                   REGION "SOLID RED"
                       IF #animation = #anSolidRed THEN
                           CASE #j OF
                               #"Part 01":
                                   #stackLight := #stackLight OR #"Part 01 Red On";
                                   #stackLight := #stackLight AND (NOT #"Part 01 Yellow On");
                                   #stackLight := #stackLight AND (NOT #"Part 01 Green On");
                               #"Part 02":
                                   #stackLight := #stackLight OR #"Part 02 Red On";
                                   #stackLight := #stackLight AND (NOT #"Part 02 Yellow On");
                                   #stackLight := #stackLight AND (NOT #"Part 02 Green On");
                               #"Part 03":
                                   #stackLight := #stackLight OR #"Part 03 Red On";
                                   #stackLight := #stackLight AND (NOT #"Part 03 Yellow On");
                                   #stackLight := #stackLight AND (NOT #"Part 03 Green On");
                               #"Part 04":
                                   #stackLight := #stackLight OR #"Part 04 Red On";
                                   #stackLight := #stackLight AND (NOT #"Part 04 Yellow On");
                                   #stackLight := #stackLight AND (NOT #"Part 04 Green On");
                               #"Part 05":
                                   #stackLight := #stackLight OR #"Part 05 Red On";
                                   #stackLight := #stackLight AND (NOT #"Part 05 Yellow On");
                                   #stackLight := #stackLight AND (NOT #"Part 05 Green On");
                               #"Part 06":
                                   #stackLight := #stackLight OR #"Part 06 Red On";
                                   #stackLight := #stackLight AND (NOT #"Part 06 Yellow On");
                                   #stackLight := #stackLight AND (NOT #"Part 06 Green On");
                               ELSE
                                   ;
                           END_CASE;
                       END_IF;
                   END_REGION

                   REGION "FLASHING RED"
                       IF #animation = #anFlashRed THEN

                           REGION "RED ON"
                               IF "Clock_1Hz" THEN
                                   CASE #j OF
                                       #"Part 01":
                                           #stackLight := #stackLight OR #"Part 01 Red On";
                                           #stackLight := #stackLight AND (NOT #"Part 01 Yellow On");
                                           #stackLight := #stackLight AND (NOT #"Part 01 Green On");
                                       #"Part 02":
                                           #stackLight := #stackLight OR #"Part 02 Red On";
                                           #stackLight := #stackLight AND (NOT #"Part 02 Yellow On");
                                           #stackLight := #stackLight AND (NOT #"Part 02 Green On");
                                       #"Part 03":
                                           #stackLight := #stackLight OR #"Part 03 Red On";
                                           #stackLight := #stackLight AND (NOT #"Part 03 Yellow On");
                                           #stackLight := #stackLight AND (NOT #"Part 03 Green On");
                                       #"Part 04":
                                           #stackLight := #stackLight OR #"Part 04 Red On";
                                           #stackLight := #stackLight AND (NOT #"Part 04 Yellow On");
                                           #stackLight := #stackLight AND (NOT #"Part 04 Green On");
                                       #"Part 05":
                                           #stackLight := #stackLight OR #"Part 05 Red On";
                                           #stackLight := #stackLight AND (NOT #"Part 05 Yellow On");
                                           #stackLight := #stackLight AND (NOT #"Part 05 Green On");
                                       #"Part 06":
                                           #stackLight := #stackLight OR #"Part 06 Red On";
                                           #stackLight := #stackLight AND (NOT #"Part 06 Yellow On");
                                           #stackLight := #stackLight AND (NOT #"Part 06 Green On");
                                       ELSE
                                           ;
                                   END_CASE;
                               END_IF;
                           END_REGION

                           REGION "RED OFF"
                               IF NOT "Clock_1Hz" THEN
                                   CASE #j OF
                                       #"Part 01":
                                           #stackLight := #stackLight AND (NOT #"Part 01 Red On");
                                           #stackLight := #stackLight AND (NOT #"Part 01 Yellow On");
                                           #stackLight := #stackLight AND (NOT #"Part 01 Green On");
                                       #"Part 02":
                                           #stackLight := #stackLight AND (NOT #"Part 02 Red On");
                                           #stackLight := #stackLight AND (NOT #"Part 02 Yellow On");
                                           #stackLight := #stackLight AND (NOT #"Part 02 Green On");
                                       #"Part 03":
                                           #stackLight := #stackLight AND (NOT #"Part 03 Red On");
                                           #stackLight := #stackLight AND (NOT #"Part 03 Yellow On");
                                           #stackLight := #stackLight AND (NOT #"Part 03 Green On");
                                       #"Part 04":
                                           #stackLight := #stackLight AND (NOT #"Part 04 Red On");
                                           #stackLight := #stackLight AND (NOT #"Part 04 Yellow On");
                                           #stackLight := #stackLight AND (NOT #"Part 04 Green On");
                                       #"Part 05":
                                           #stackLight := #stackLight AND (NOT #"Part 05 Red On");
                                           #stackLight := #stackLight AND (NOT #"Part 05 Yellow On");
                                           #stackLight := #stackLight AND (NOT #"Part 05 Green On");
                                       #"Part 06":
                                           #stackLight := #stackLight AND (NOT #"Part 06 Red On");
                                           #stackLight := #stackLight AND (NOT #"Part 06 Yellow On");
                                           #stackLight := #stackLight AND (NOT #"Part 06 Green On");
                                       ELSE
                                           ;
                                   END_CASE;
                               END_IF;
                           END_REGION

                       END_IF;
                   END_REGION

                   REGION "COPY OUT TO GLOBAL"
                       #stations.current[#i].stackLightOut := #stackLight;
                   END_REGION

               END_FOR;
           END_REGION

       END_FOR;
   END_REGION
END_FUNCTION_BLOCK

FUNCTION_BLOCK "KP8 Button Activation"   // FB12, SCL
{ S7_Optimized_Access := 'TRUE' }
VERSION : 0.1
   VAR_INPUT
      constants : "Constants";
   END_VAR
   VAR_IN_OUT
      stations : "Stations";
   END_VAR
   VAR_TEMP
      btnCount : Int;
      currentPNs : Array[0..7] of WString[40];
      i : Int;
      init : Bool;
      j : Int;
      stnCount : Int;
      temp : Int;
   END_VAR
BEGIN
   REGION "GET STATION COUNT"
       #stnCount := #constants.stationCount - 1;
       #btnCount := #constants.buttonCount - 1;
   END_REGION

   REGION "LOOP THROUGH STATIONS"
       FOR #i := 0 TO #stnCount DO

           #currentPNs := #stations.current[#i].partNumbers;

           REGION "LOOP THROUGH BUTTONS"
               FOR #j := 0 TO #btnCount DO

                       REGION "ACTIVATE BUTTON"
                           IF LEN(#currentPNs[#j]) <> 0 THEN
                               #stations.current[#i].kp8Config.activate[#j] := TRUE;
                               #stations.current[#i].kp8Config.colorOff[#j] := 'green';
                               #stations.current[#i].kp8Config.colorOn1[#j] := 'yellow';
                               #stations.current[#i].kp8Config.colorOn2[#j] := '';
                               #stations.current[#i].kp8Config.flash[#j] := FALSE;
                               #stations.current[#i].kp8Config.group[#j] := 0;
                               #stations.current[#i].kp8Config.mode[#j] := TRUE;
                           END_IF;
                       END_REGION

                       REGION "DEACTIVATE BUTTON"
                           IF LEN(#currentPNs[#j]) = 0 THEN
                               #stations.current[#i].kp8Config.activate[#j] := FALSE;
                               #stations.current[#i].kp8Config.colorOff[#j] := '';
                               #stations.current[#i].kp8Config.colorOn1[#j] := '';
                               #stations.current[#i].kp8Config.colorOn2[#j] := '';
                               #stations.current[#i].kp8Config.flash[#j] := FALSE;
                               #stations.current[#i].kp8Config.group[#j] := 0;
                               #stations.current[#i].kp8Config.mode[#j] := FALSE;
                           END_IF;
                       END_REGION

               END_FOR;
           END_REGION

           REGION "SOFT INIT"
               IF #stations.current[#i].kp8Config <> #stations.old[#i].kp8Config THEN
                   #stations.current[#i].init.soft := TRUE;
               END_IF;
           END_REGION

       END_FOR;
   END_REGION
END_FUNCTION_BLOCK

FUNCTION_BLOCK "Remove Part Request"   // FB13, SCL
{ S7_Optimized_Access := 'TRUE' }
VERSION : 0.1
   VAR_INPUT
      constants : "Constants";
   END_VAR
   VAR_IN_OUT
      pRow : Int;
      requests : "Part Request Data";
      stations : "Stations";
   END_VAR
   VAR_TEMP
      address : UInt;
      blankRow : "Table Row";
      hasPart : Bool;
      i : Int;
      j : Int;
      k : Int;
      logAddress : UInt;
      maxRows : Int;
      noPart : Bool;
      oldPartReq : Bool;
      partNumber : WString;
      partReq : Bool;
      pRemoveRow : Int;
      btnCount : Int;
      stnCount : Int;
      removeAddress : Bool;
   END_VAR
BEGIN
   REGION "COPY TO LOCAL"
       #maxRows := #constants.partReqRows - 1;
       #stnCount := #constants.stationCount - 1;
       #btnCount := #constants.buttonCount - 1;
   END_REGION


   REGION "LOOP THROUGH STATIONS"
       FOR #i := 0 TO #stnCount DO

           REGION "LOOP THROUGH BUTTONS"
               FOR #j := 1 TO #btnCount DO

                   REGION "PRE-CONDITION"
                       // copy bits for falling edge detection
                       #partReq := #stations.current[#i].btnStates[#j];
                       #oldPartReq := #stations.old[#i].btnStates[#j];
                   END_REGION

                   REGION "DETERMINE STATE"
                       // falling edge detection
                       IF NOT #partReq AND #oldPartReq THEN
                           // copy to local
                           #partNumber := #stations.current[#i].partNumbers[#j];
                           // no part
                           IF #partNumber = wstring#'' THEN
                               #hasPart := FALSE;
                               #noPart := TRUE;
                           END_IF;
                           // has part
                           IF #partNumber <> wstring#'' THEN
                               #hasPart := TRUE;
                               #noPart := FALSE;
                           END_IF;
                       END_IF;
                   END_REGION

                   REGION "NO PART"
                       IF #noPart THEN
                           // turn off the lights
                           #hasPart := FALSE;
                           #noPart := FALSE;
                       END_IF;

                   END_REGION

                   REGION "HAS PART"
                       IF #hasPart THEN
                           // turn off the lights
                           #hasPart := FALSE;
                           // calculate address
                           #address := (INT_TO_UINT(#i) + 1) * 10 + (INT_TO_UINT(#j) + 1);
                           // precondition remove address flag
                           #removeAddress := FALSE;
                           // check table for previous entry
                           FOR #k := 0 TO #maxRows DO
                               #logAddress := #requests.row[#k].address;
                               // remove matching address flag
                               IF #logAddress = #address THEN
                                   #removeAddress := TRUE;
                                   #pRemoveRow := #k;
                               END_IF;
                           END_FOR;
                       END_IF;
                   END_REGION

                   REGION "REMOVE ADDRESS"
                       IF #removeAddress THEN

                           // turn off the lights
                           #removeAddress := FALSE;

                           REGION "REMOVAL PROCESS"
                               #requests.row[#pRemoveRow] := #blankRow;
                           END_REGION

                           REGION "ADJUST TABLE BLANK ROW POINTER"
                               // decriment row pointer
                               #pRow := #pRow - 1;
                               IF #pRow < 0 THEN
                                   #pRow := 0;
                               END_IF;
                           END_REGION

                       END_IF;
                   END_REGION

               END_FOR;

           END_REGION

       END_FOR;
   END_REGION
END_FUNCTION_BLOCK

FUNCTION_BLOCK "HMI Settings Screen"   // FB14, LAD
{ S7_Optimized_Access := 'TRUE' }
VERSION : 0.1
   VAR_INPUT
      constants : "Constants";
   END_VAR
   VAR_IN_OUT
      settings : "Settings Screen";
      stations : "Stations";
   END_VAR
   VAR
      tmrTimeOut : TON_TIME;
      instStaSel : "Station Selection";
      instKP8BtnSel : "KP8 Button Selections";
      instStnDetails : "Station Details";
   END_VAR
   VAR CONSTANT
      ptTimeOut : Time := t#15m;
   END_VAR
BEGIN

REGION Network 1: ENTRY TIMEOUT
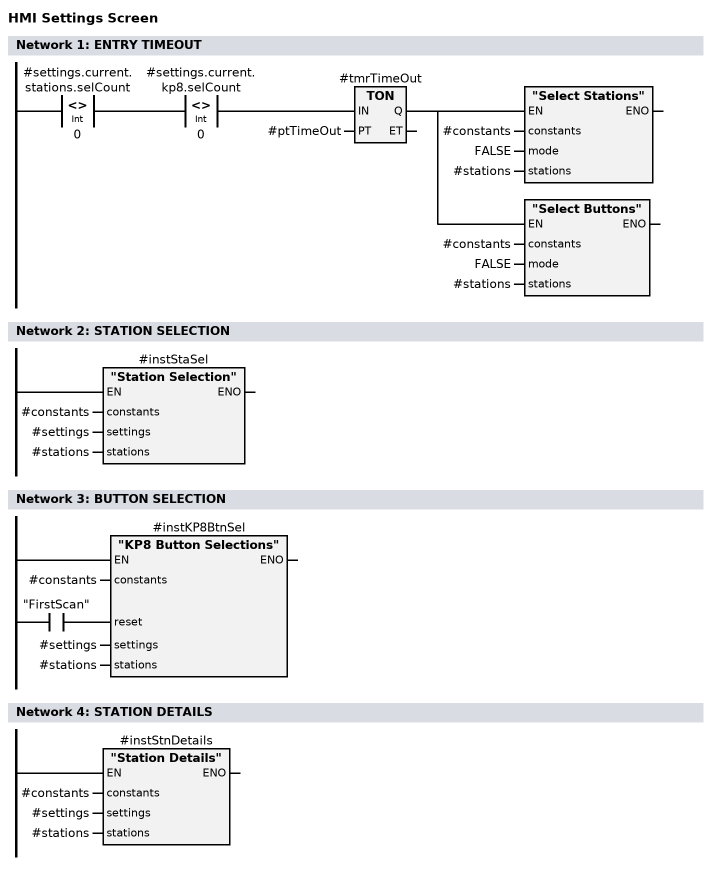
   #tmrTimeOut(IN := (#settings.current.stations.selCount <> 0) AND (#settings.current.kp8.selCount <> 0),   // TON
               PT := #ptTimeOut);
   IF #tmrTimeOut.Q THEN
       "Select Stations"(constants := #constants, mode := FALSE, stations := #stations);
       "Select Buttons"(constants := #constants, mode := FALSE, stations := #stations);
   END_IF;
END_REGION

REGION Network 2: STATION SELECTION
   RUNG wire#powerrail
      #instStaSel(constants := #constants, settings := #settings, stations := #stations)
   END_RUNG
   // the same network as SCL:
   #instStaSel(constants := #constants, settings := #settings, stations := #stations);   // "Station Selection"
END_REGION

REGION Network 3: BUTTON SELECTION
   RUNG wire#powerrail
      #instKP8BtnSel(reset := wire#w1, constants := #constants, settings := #settings, stations := #stations)
   END_RUNG
   RUNG wire#powerrail
      Contact( "FirstScan" )
   END_RUNG wire#w1
   // the same network as SCL:
   #instKP8BtnSel(constants := #constants, reset := "FirstScan", settings := #settings, stations := #stations);   // "KP8 Button Selections"
END_REGION

REGION Network 4: STATION DETAILS
   RUNG wire#powerrail
      #instStnDetails(constants := #constants, settings := #settings, stations := #stations)
   END_RUNG
   // the same network as SCL:
   #instStnDetails(constants := #constants, settings := #settings, stations := #stations);   // "Station Details"
END_REGION
END_FUNCTION_BLOCK

FUNCTION_BLOCK "Collapse Table"   // FB15, SCL
{ S7_Optimized_Access := 'TRUE' }
VERSION : 0.1
   VAR_INPUT
      constants : "Constants";
   END_VAR
   VAR_IN_OUT
      requests : "Part Request Data";
   END_VAR
   VAR
      tableBox : "Part Request Data";
   END_VAR
   VAR_TEMP
      blankRow : "Table Row";
      collapseReq : Bool;
      i : Int;
      maxRows : Int;
      pCollapse : Int;
   END_VAR
BEGIN
   REGION "COPY TO LOCAL"
       #maxRows := #constants.partReqRows - 1;
   END_REGION

   REGION "REMOVE EMPTY ROWS"
       FOR #i := 0 TO #maxRows DO

           REGION "ROW IS NOT EMPTY"
               IF #requests.row[#i].address <> 0 THEN

                   REGION "MOVE TO TEMP TABLE"
                       #tableBox.row[#pCollapse] := #requests.row[#i];
                   END_REGION

                   REGION "POINTERS AND FLAGS"
                       #pCollapse := #pCollapse + 1;
                       #collapseReq := TRUE;
                   END_REGION

               END_IF;
           END_REGION

       END_FOR;
   END_REGION

   REGION "COLLAPSE TABLE"
       IF #collapseReq THEN

           REGION "TURN OFF THE LIGHTS"
               #collapseReq := FALSE;
           END_REGION

           REGION "COPY TEMP TO PERMANENT"
               #requests := #tableBox;
           END_REGION

           REGION "CLEAR VALUES FROM TEMP TABLE"
               FOR #i := 0 TO #maxRows DO
                   #tableBox.row[#i] := #blankRow;
               END_FOR;
           END_REGION
       END_IF;

   END_REGION
END_FUNCTION_BLOCK

FUNCTION_BLOCK "HMI Populate Part Call"   // FB16, SCL
{ S7_Optimized_Access := 'TRUE' }
VERSION : 0.1
   VAR_INPUT
      constants : "Constants";
      requests : "Part Request Data";
   END_VAR
   VAR_IN_OUT
      partCall : "Part Call Screen";
   END_VAR
   VAR
      pDisplay : Int;
   END_VAR
   VAR_TEMP
      firstRow : Int;
      i : Int;
      lastRow : Int;
      maxRows : Int;
      pRow : Int;
      visibleRows : Int;
      thisRow : Int;
   END_VAR
BEGIN
   #visibleRows := #constants.hmiRowCount - 1;
   #maxRows := #constants.partReqRows - 1;
   #firstRow := 0;
   #lastRow := #firstRow + #visibleRows;

   FOR #i := 0 TO #visibleRows DO
       #partCall.current[#i] := #requests.row[#i];
   END_FOR;
END_FUNCTION_BLOCK

FUNCTION_BLOCK "Clear Part Requests"   // FB17, SCL
{ S7_Optimized_Access := 'TRUE' }
VERSION : 0.1
   VAR_INPUT
      constants : "Constants";
      clearRequest : Bool;
   END_VAR
   VAR_IN_OUT
      requests : "Part Request Data";
      partCall : "Part Call Screen";
   END_VAR
   VAR_TEMP
      blankRow : "Table Row";
      i : Int;
      maxRows : Int;
   END_VAR
BEGIN
   REGION "ON REQUEST"
       IF #clearRequest THEN

           REGION "CLEAR HMI TABLE"
               #maxRows := #constants.hmiRowCount - 1;
               FOR #i := 0 TO #maxRows DO
                   #partCall.current[#i] := #blankRow;
               END_FOR;
           END_REGION

           REGION "CLEAR PART REQUEST DATA BASE"
               #maxRows := #constants.partReqRows - 1;
               FOR #i := 0 TO #maxRows DO
                   #requests.row[#i] := #blankRow;
               END_FOR;
           END_REGION

       END_IF;
   END_REGION
END_FUNCTION_BLOCK

FUNCTION_BLOCK "Load Default Timer Presets"   // FB18, SCL
{ S7_Optimized_Access := 'TRUE' }
VERSION : 0.1
   VAR_INPUT
      constants : "Constants";
      req : Bool;
   END_VAR
   VAR_IN_OUT
      stations : "Stations";
   END_VAR
   VAR
      oldReq : Bool;
   END_VAR
   VAR_TEMP
      alotted : Real;
      btnCount : Int;
      critical : Real;
      i : Int;
      j : Int;
      stnCount : Int;
      partNumber : WString;
   END_VAR
BEGIN
   REGION "COPY TO LOCAL"
       #alotted := #constants.defaultAlotted;
       #btnCount := #constants.buttonCount - 1;
       #critical := #constants.defaultCritical;
       #stnCount := #constants.stationCount - 1;
   END_REGION

   REGION "ON REQUEST RISING EDGE"
       IF #req AND NOT #oldReq THEN

           REGION "LOOP THROUGH STATIONS" 
               FOR #i := 0 TO #stnCount DO

                   REGION "LOOP THROUGH BUTTONS"
                       FOR #j := 0 TO #btnCount DO

                           REGION "IF BUTTON HAS ASSOCIATED PN"
                               #partNumber := #stations.current[#i].partNumbers[#j];
                               IF LEN(#partNumber) <> 0 THEN

                                   REGION "ASSIGN PRESET VALUES"
                                       #stations.current[#i].presetTime.allotted[#j] := #alotted;
                                       #stations.current[#i].presetTime.critical[#j] := #critical;
                                   END_REGION

                               END_IF;
                           END_REGION

                       END_FOR;
                   END_REGION

               END_FOR;
           END_REGION

       END_IF;
   END_REGION

   REGION "CHANGE DETECTION"
       #oldReq := #req;
   END_REGION ;
END_FUNCTION_BLOCK

FUNCTION_BLOCK "LED Populate Sign"   // FB19, SCL
{ S7_Optimized_Access := 'TRUE' }
VERSION : 0.1
   VAR_INPUT
      constants : "Constants";
      requests : "Part Request Data";
   END_VAR
   VAR_IN_OUT
      ledData : "LED Sign Data";
   END_VAR
   VAR_TEMP
      i : Int;
      visibleRows : Int;
   END_VAR
BEGIN
   REGION "COPY TO LOCAL"
       #visibleRows := #constants.ledRowCount - 1;
   END_REGION

   REGION "POPULATE SIGN DATA"
       FOR #i := 0 TO #visibleRows DO
           #ledData.row[#i] := #requests.row[#i];
       END_FOR;
   END_REGION
END_FUNCTION_BLOCK

FUNCTION_BLOCK "Station Selection"   // FB20, SCL
{ S7_Optimized_Access := 'TRUE' }
VERSION : 0.1
   VAR_INPUT
      constants : "Constants";
   END_VAR
   VAR_IN_OUT
      settings : "Settings Screen";
      stations : "Stations";
   END_VAR
   VAR
      firstStn : Int;
      rt : "Runtime Data";
      selectionExe : Bool;
      old : Struct
         prevGrp : Bool;
         nextGrp : Bool;
         stnSlct : Array[0..11] of Bool;
      END_STRUCT;
   END_VAR
   VAR_TEMP
      animate : USInt;
      btnPress : Bool;
      count : Int;
      currentBtn : Bool;
      evalObjCount : Int;
      i : Int;
      oldBtn : Bool;
      pStn : Int;
      stnCount : Int;
      stnName : WString;
      stnSelected : Bool;
      selState : Bool;
      timerExpired : Bool;
      stnSelLblCount : Int;
   END_VAR
   VAR CONSTANT
      ptTimer : Real := 1.5;
   END_VAR
BEGIN
   REGION "UI INTERACTION ANIMATIONS"

       REGION "NEXT GROUP"
           #btnPress := #settings.current.stations.nextGroup.actuate;
           #animate := "Animate Bool"(colorTrue := #constants.colorLib.BgLGr,
                                      colorFalse := #constants.colorLib.BgGray,
                                      evalSignal := #btnPress);
           #settings.current.stations.nextGroup.animate := #animate;
       END_REGION

       REGION "PREVIOUS GROUP"
           #btnPress := #settings.current.stations.prevGroup.actuate;
           #animate := "Animate Bool"(colorTrue := #constants.colorLib.BgLGr,
                                      colorFalse := #constants.colorLib.BgGray,
                                      evalSignal := #btnPress);
           #settings.current.stations.prevGroup.animate := #animate;
       END_REGION

       REGION "SELECT ALL STATIONS"
           #btnPress := #settings.current.stations.selectAll.actuate;
           #animate := "Animate Bool"(colorTrue := #constants.colorLib.BgLGr,
                                      colorFalse := #constants.colorLib.BgGray,
                                      evalSignal := #settings.current.stations.selectAll.actuate);
           #settings.current.stations.selectAll.animate := #animate;
       END_REGION

   END_REGION

   REGION "POPULATE STATION LABELS"

       REGION "PROCESS NEXT GROUP PRESS"

           REGION "COPY TO LOCAL"
               #stnCount := #constants.stationCount - 1;
               #currentBtn := #settings.current.stations.nextGroup.actuate;
               #oldBtn := #old.nextGrp;
           END_REGION

           REGION "FALLING EDGE OF NEXT GROUP"
               IF NOT #currentBtn AND #oldBtn THEN

                   REGION "INCREMENT FIRST STATION"
                       #firstStn := #firstStn + 2;
                   END_REGION

                   REGION "UPPER LIMIT ROLL OVER"
                       IF #firstStn > #stnCount THEN
                           #firstStn := #firstStn - #stnCount - 1;
                       END_IF;
                   END_REGION

               END_IF;
           END_REGION

           REGION "NEXT GROUP CHANGE DETECTION"
               #old.nextGrp := #currentBtn;
           END_REGION

       END_REGION

       REGION "PROCESS PREVIOUS GROUP PRESS"

           REGION "COPY TO LOCAL"
               #currentBtn := #settings.current.stations.prevGroup.actuate;
               #oldBtn := #old.prevGrp;
               #stnCount := #constants.stationCount - 1;
           END_REGION

           REGION "FALLING EDGE OF PREVIOUS GROUP"
               IF NOT #currentBtn AND #oldBtn THEN

                   REGION "DECREMENT FIRST STATION"
                       #firstStn := #firstStn - 2;
                   END_REGION

                   REGION "LOWER LIMIT ROLL OVER"
                       IF #firstStn < 0 THEN
                           #firstStn := #firstStn + #stnCount + 1;
                       END_IF;
                   END_REGION

               END_IF;
           END_REGION

           REGION "PREVIOUS GROUP CHANGE DETECTION"
               #old.prevGrp := #currentBtn;
           END_REGION

       END_REGION

       REGION "WRITE LABEL"

           REGION "COPY TO LOCAL"
               #evalObjCount := #constants.hmiSelStnCount - 1;
               #stnCount := #constants.stationCount - 1;
           END_REGION

           REGION "FOR EACH STATION SELECTION BUTTON"
               FOR #i := 0 TO #evalObjCount DO

                   REGION "CALCULATE POINTER"
                       #pStn := #firstStn + #i;
                   END_REGION

                   REGION "UPPER LIMIT ROLL OVER"
                       IF #pStn > #stnCount THEN
                           #pStn := #firstStn + #i - #stnCount - 1;
                       END_IF;
                   END_REGION

                   REGION "BUILD NAME"
                       #stnName := CONCAT_WSTRING(IN1 := #stations.current[#pStn].line,
                                                  IN2 := wstring#' ',
                                                  IN3 := "Strip Sign"(USINT_TO_WSTRING(#stations.current[#pStn].dropZone)));
                   END_REGION

                   REGION "WRITE NAME"
                       #settings.current.stations.selectBtns[#i].label := #stnName;
                   END_REGION

               END_FOR;
           END_REGION

       END_REGION

   END_REGION

   REGION "SINGLE STATION SELECTION"

       REGION "COPY TO LOCAL"
           #stnSelLblCount := #constants.hmiSelStnCount - 1;
       END_REGION

       REGION "LOOP THROUGH DISPLAYED STATIONS"
           FOR #i := 0 TO #stnSelLblCount DO

               REGION "CALCULATE POINTER"
                   #pStn := #firstStn + #i;
               END_REGION

               REGION "UPPER LIMIT ROLL OVER"
                   #stnCount := #constants.stationCount - 1;
                   IF #pStn > #stnCount THEN
                       #pStn := #firstStn + #i - #stnCount - 1;
                   END_IF;
               END_REGION

               REGION "COPY TO LOCAL"
                   #currentBtn := #settings.current.stations.selectBtns[#i].actuate;
                   #oldBtn := #old.stnSlct[#i];
               END_REGION

               REGION "TOGGLE STATE ON FALLING EDGE"
                   IF NOT #currentBtn AND #oldBtn THEN
                       #selState := #stations.current[#pStn].settings.selected;
                       #selState := NOT #selState;
                       #stations.current[#pStn].settings.selected := #selState;
                   END_IF;
               END_REGION

               REGION "STATION SELECTION CHANGE DETECTION"
                   #old.stnSlct[#i] := #currentBtn;
               END_REGION

           END_FOR;
       END_REGION

   END_REGION

   REGION "MULTI SELECT TIMER"

       REGION "RUNTIME CALL"
           #rt.elapsed := RUNTIME(#rt.mem);
       END_REGION

       REGION "TIMER"

           REGION "COPY TO LOCAL"
               #btnPress := #settings.current.stations.selectAll.actuate;
           END_REGION

           REGION "ACCUMULATE RT VALUES"
               IF #btnPress THEN
                   #rt.asReal += LREAL_TO_REAL(#rt.elapsed);
               END_IF;
           END_REGION

           REGION "SET TIMER FLAG"
               IF #rt.asReal < #ptTimer THEN
                   #timerExpired := FALSE;
               END_IF;
               IF #rt.asReal >= #ptTimer THEN
                   #timerExpired := TRUE;
                   #rt.asReal := 0.0;
               END_IF;
           END_REGION

           REGION "RESET ACCUMULATED VALUE"
               IF NOT #btnPress THEN
                   #rt.asReal := 0.0;
                   #selectionExe := FALSE;
               END_IF;
           END_REGION

       END_REGION

   END_REGION

   REGION "EVALUATE MULTI SELECTION"
       IF #timerExpired AND NOT #selectionExe THEN

           REGION "COPY TO LOCAL"
               #stnCount := #settings.current.stations.selCount;
           END_REGION

           REGION "SELECT ALL"
               IF #stnCount < #constants.stationCount THEN
                   "Select Stations"(constants := #constants,
                                     mode := TRUE,
                                     stations := #stations);
               END_IF;
           END_REGION

           REGION "DESELECT ALL"
               IF #stnCount = #constants.stationCount THEN
                   "Select Stations"(constants := #constants,
                                     mode := FALSE,
                                     stations := #stations);
               END_IF;
           END_REGION

           REGION "FLAG SELECTION EXECUTED"
               #selectionExe := TRUE;
           END_REGION

       END_IF;
   END_REGION

   REGION "SELECTION ANIMATIONS"

       REGION "COPY TO LOCAL"
           #stnSelLblCount := #constants.hmiSelStnCount - 1;
           #stnCount := #constants.stationCount - 1;
       END_REGION

       REGION "LOOP THROUGH BUTTONS"
           FOR #i := 0 TO #stnSelLblCount DO

               REGION "CALCULATE POINTER"
                   #pStn := #firstStn + #i;
               END_REGION

               REGION "UPPER LIMIT ROLL OVER"
                   IF #pStn > #stnCount THEN
                       #pStn := #firstStn + #i - #stnCount - 1;
                   END_IF;
               END_REGION

               REGION "COPY TO LOCAL"
                   #currentBtn := #settings.current.stations.selectBtns[#i].actuate;
                   #stnSelected := #stations.current[#pStn].settings.selected;
               END_REGION

               REGION "DRAW SELCTION HIGHLIGHTS"
                   #animate := "Animate Bool"(colorTrue := #constants.colorLib.BgLTe,
                                              colorFalse := #constants.colorLib.BgGray,
                                              evalSignal := #stnSelected);
               END_REGION

               REGION "ANIMATE BUTTON PRESS"
                   #animate := "Animate Bool"(colorTrue := #constants.colorLib.BgDTe,
                                              colorFalse := #animate,
                                              evalSignal := #currentBtn);
                   #settings.current.stations.selectBtns[#i].animate := #animate;
               END_REGION

           END_FOR;
       END_REGION

   END_REGION

   REGION "COUNT SELECTED STATIONS"

       REGION "INITIALIZE LOCAL"
           #count := 0;
           #evalObjCount := #constants.stationCount - 1;
       END_REGION

       REGION "LOOP THROUGH STATIONS"
           FOR #i := 0 TO #evalObjCount DO

               REGION "INCREMENT COUNT ON SELECTION"
                   #stnSelected := #stations.current[#i].settings.selected;
                   IF #stnSelected THEN
                       #count += 1;
                   END_IF;
               END_REGION

           END_FOR;
       END_REGION

       REGION "SAVE COUNT"
           #settings.current.stations.selCount := #count;
       END_REGION

   END_REGION
END_FUNCTION_BLOCK

FUNCTION_BLOCK "KP8 Button Selections"   // FB21, SCL
{ S7_Optimized_Access := 'TRUE' }
VERSION : 0.1
   VAR_INPUT
      constants : "Constants";
      reset : Bool;
   END_VAR
   VAR_IN_OUT
      settings : "Settings Screen";
      stations : "Stations";
   END_VAR
   VAR
      enableState : Bool;
      oldBtnPresses : Array[0..7] of Bool;
      oldSelState : Array[0..7] of Bool;
      oldSelStnCount : Int;
      rt : "Runtime Data";
      timerExpired : Bool;
      selectionExe : Bool;
   END_VAR
   VAR_TEMP
      animate : USInt;
      btnCount : Int;
      btnPress : Bool;
      count : Int;
      i : Int;
      j : Int;
      mode : Bool;
      oldPress : Bool;
      pBtn : Int;
      selBtnCount : Int;
      selStnCount : Int;
      stnCount : Int;
      stnSelected : Bool;
   END_VAR
   VAR CONSTANT
      selectAllTime : Real := 1.5;
   END_VAR
BEGIN
   REGION "ENABLE KP8 BUTTON ASSIGNMENT SECTION"

       REGION "ENABLE"

           REGION "COPY TO LOCAL"
               #selStnCount := #settings.current.stations.selCount;
           END_REGION

           REGION "ON CHANGE IN SELECTED STATION COUNT"
               IF #selStnCount <> 0 AND #selStnCount <> #oldSelStnCount THEN

                   REGION "ENABLE KP8 SELECTIONS"
                       #enableState := TRUE;
                   END_REGION

               END_IF;
           END_REGION

       END_REGION

       REGION "DISABLE"

           REGION "COPY TO LOCAL"
               #selStnCount := #settings.current.stations.selCount;
               #btnCount := #constants.buttonCount - 1;
           END_REGION

           REGION "ON DESELETION OF LAST STATION"
               IF #selStnCount = 0 AND #selStnCount <> #oldSelStnCount THEN

                   REGION "RESET ENABLED STATE"
                       #enableState := FALSE;
                   END_REGION

                   REGION "RESET BUTTON SELECTION STATES"
                       FOR #i := 0 TO #btnCount DO
                           #settings.current.kp8.btnSelState[#i] := FALSE;
                       END_FOR;
                   END_REGION

               END_IF;
           END_REGION

       END_REGION

   END_REGION

   REGION "SINGLE BUTTON SELECTION"

       REGION "COPY TO LOCAL"
           #btnCount := #constants.buttonCount - 1;
       END_REGION

       REGION "LOOP THROUGH BUTTONS"
           FOR #i := 0 TO #btnCount DO

               REGION "EXCLUDE STOP RUNTIME AND RESET SELECTED BUTTONS"
                   IF #i <> 0 AND #i <> 4 THEN

                       REGION "COPY TO LOCAL"

                           REGION "CALCULATE BUTTON POINTER"
                               CASE #i OF
                                   1:
                                       #pBtn := 5;
                                   2:
                                       #pBtn := 3;
                                   3:
                                       #pBtn := 1;
                                   5:
                                       #pBtn := 4;
                                   6:
                                       #pBtn := 2;
                                   7:
                                       #pBtn := 0;
                                   ELSE
                                       ;
                               END_CASE;

                           END_REGION

                           #btnPress := #settings.current.kp8.buttons[#i].actuate OR #settings.current.viewingStation.btns[#pBtn].select.actuate;
                           #oldPress := #oldBtnPresses[#i];

                       END_REGION

                       REGION "TOGGLE STATE ON FALLING EDGE"
                           IF NOT #btnPress AND #oldPress THEN
                               #settings.current.kp8.btnSelState[#i] := NOT #settings.current.kp8.btnSelState[#i];
                               #settings.current.kp8.selBtnNumber := #i;
                           END_IF;
                       END_REGION

                       REGION "SAVE SELECTED BUTTON NUMBER ON DESELECT"
                           IF NOT #settings.current.kp8.btnSelState[#i] AND #oldSelState[#i] THEN
                               FOR #j := 0 TO #btnCount DO
                                   IF #settings.current.kp8.btnSelState[#j] THEN
                                       #settings.current.kp8.selBtnNumber := #j;
                                   END_IF;
                               END_FOR;
                           END_IF;
                       END_REGION

                       REGION "KP8 BUTON SELECTION CHANGE DETECTION"
                           #oldBtnPresses[#i] := #btnPress;
                       END_REGION

                   END_IF;
               END_REGION

           END_FOR;
       END_REGION

   END_REGION

   REGION "MULTI BUTTON SELECTION"

       REGION "MULTI SELECT TIMER"

           REGION "RUNTIME CALL"
               #rt.elapsed := RUNTIME(#rt.mem);
           END_REGION

           REGION "TIMER"

               REGION "COPY TO LOCAL"
                   #btnPress := #settings.current.kp8.selectButtons.actuate;
               END_REGION

               REGION "ACCUMULATE RT VALUES"
                   IF #btnPress THEN
                       #rt.asReal += LREAL_TO_REAL(#rt.elapsed);
                   END_IF;
               END_REGION

               REGION "SET TIMER FLAG"
                   IF #rt.asReal < #selectAllTime THEN
                       #timerExpired := FALSE;
                   END_IF;
                   IF #rt.asReal >= #selectAllTime THEN
                       #timerExpired := TRUE;
                       #rt.asReal := 0.0;
                   END_IF;
               END_REGION

               REGION "RESET ACCUMULATED VALUE"
                   IF NOT #btnPress THEN
                       #rt.asReal := 0.0;
                       #selectionExe := FALSE;
                   END_IF;
               END_REGION

           END_REGION

       END_REGION

       REGION "EVALUATE MULTI SELECTION"
           IF #timerExpired AND NOT #selectionExe THEN

               REGION "COPY TO LOCAL"
                   #btnCount := #constants.buttonCount - 1;
                   #selBtnCount := #settings.current.kp8.selCount;
               END_REGION

               REGION "SELECT ALL"
                   IF #selBtnCount < #btnCount - 1 THEN
                       #mode := TRUE;
                   END_IF;
               END_REGION

               REGION "DESELECT ALL"
                   IF #selBtnCount = #btnCount - 1 THEN
                       #mode := FALSE;
                   END_IF;
               END_REGION

               REGION "SAVE SELECTIONS"
                   FOR #i := 0 TO #btnCount DO

                       REGION "EXCLUDE STOP RUNTIME AND RESET SELECTED BUTTONS"
                           IF #i <> 0 AND #i <> 4 THEN

                               REGION "PERFROM SELECTION"
                                   #settings.current.kp8.btnSelState[#i] := #mode;
                               END_REGION

                           END_IF;
                       END_REGION

                   END_FOR;
               END_REGION

               REGION "SET SELECED BUTTON NUMBER TO 1"
                   #settings.current.kp8.selBtnNumber := 0;
               END_REGION

               REGION "FLAG SELECTION EXECUTED"
                   #selectionExe := TRUE;
               END_REGION

           END_IF;
       END_REGION
   END_REGION

   REGION "SAVE BUTTON SELECTIONS TO STATIONS"

       REGION "COPY TO LOCAL"
           #selStnCount := #settings.current.stations.selCount;
       END_REGION

       REGION "ON CHANGE IN BUTTON OR STATION SELECTON"
           IF #settings.current.kp8.btnSelState <> #oldSelState OR #selStnCount <> #oldSelStnCount THEN

               REGION "COPY TO LOCAL"
                   #stnCount := #constants.stationCount - 1;
               END_REGION

               REGION "FOR SELECTED STATIONS"
                   FOR #i := 0 TO #stnCount DO
                       #stnSelected := #stations.current[#i].settings.selected;
                       IF #stnSelected THEN

                           REGION "SAVE BUTTON SELECTION STATE"
                               #stations.current[#i].settings.btnSelection := #settings.current.kp8.btnSelState;
                           END_REGION

                       END_IF;
                   END_FOR;
               END_REGION

           END_IF;
       END_REGION

       REGION "SELECTED STATION COUNT CHANGE DETECTION"
           #oldSelStnCount := #selStnCount; 
       END_REGION

   END_REGION

   REGION "COUNT SELECTED BUTTONS"

       REGION "COPY TO LOCAL"
           #btnCount := #constants.buttonCount - 1;
       END_REGION 

       REGION "ON CHANGE IN BUTTON SELECTION STATES"
           IF #settings.current.kp8.btnSelState <> #oldSelState THEN

               REGION "INITIALIZE LOCAL"
                   #count := 0;
               END_REGION

               REGION "FOR EACH SELECTED BUTTON"
                   FOR #i := 0 TO #btnCount DO
                       IF #settings.current.kp8.btnSelState[#i] THEN

                           REGION "INCREMENT COUNT"
                               #count := #count + 1;
                           END_REGION

                       END_IF;
                   END_FOR;
               END_REGION

               REGION "SAVE COUNT"
                   #settings.current.kp8.selCount := #count;
               END_REGION

           END_IF;
       END_REGION

   END_REGION 

   REGION "UI INTERACTION ANIMATIONS"

       REGION "SELECT ALL BUTTONS"
           #btnPress := #settings.current.kp8.selectButtons.actuate;
           #animate := "Animate Bool"(colorTrue := #constants.colorLib.BgLGr,
                                      colorFalse := #constants.colorLib.BgGray,
                                      evalSignal := #btnPress);
           #settings.current.kp8.selectButtons.animate := #animate;
       END_REGION

       REGION "STOP RESET SELECTED STATION"
           #btnPress := #settings.current.kp8.buttons[0].actuate;
           #animate := "Animate Bool"(colorTrue := #constants.colorLib.FgGray,
                                      colorFalse := #constants.colorLib.BgGray,
                                      evalSignal := #btnPress);
           #settings.current.kp8.buttons[0].animate := #animate;
       END_REGION

       REGION "STOP RUNTIME"
           #btnPress := #settings.current.kp8.buttons[4].actuate;
           #animate := "Animate Bool"(colorTrue := #constants.colorLib.FgGray,
                                      colorFalse := #constants.colorLib.BgGray,
                                      evalSignal := #btnPress);
           #settings.current.kp8.buttons[4].animate := #animate;
       END_REGION

       REGION "BUTTON SELECTIONS"

           REGION "COPY TO LOCAL"
               #btnCount := #constants.buttonCount - 1;
           END_REGION

           REGION "FOR EACH BUTTON"     
               FOR #i := 0 TO #btnCount DO

                   REGION "EXCLUDE STOP RUNTIME AND RESET SELECTED BUTTONS"
                       IF #i <> 0 AND #i <> 4 THEN

                           REGION "ANIMATE"

                               REGION "COPY TO LOCAL"
                                   #btnPress := #settings.current.kp8.buttons[#i].actuate;
                               END_REGION

                               REGION "ENABLE/DISABLE"
                                   #animate := "Animate Bool"(colorTrue := #constants.colorLib.BgGray,
                                                              colorFalse := #constants.colorLib.disabled,
                                                              evalSignal := #enableState);
                               END_REGION

                               REGION "ENABLED SUB ANIMATIONS"
                                   IF #enableState THEN

                                       REGION "BUTTON SELECTED"
                                           #animate := "Animate Bool"(colorTrue := #constants.colorLib.BgLTe,
                                                                      colorFalse := #animate,
                                                                      evalSignal := #settings.current.kp8.btnSelState[#i]);
                                       END_REGION

                                       REGION "BUTTON UP/DOWN"
                                           #animate := "Animate Bool"(colorTrue := #constants.colorLib.BgDTe,
                                                                      colorFalse := #animate,
                                                                      evalSignal := #btnPress);
                                       END_REGION
                                   END_IF;
                               END_REGION

                               REGION "SAVE ANIMATION"
                                   #settings.current.kp8.buttons[#i].animate := #animate;
                               END_REGION

                           END_REGION

                       END_IF;
                   END_REGION

               END_FOR;
           END_REGION

       END_REGION

   END_REGION

   REGION "DRAW KP8 BUTTON LABELS"
       IF #reset THEN
           #settings.current.kp8.buttons[1].label := wstring#'6';
           #settings.current.kp8.buttons[2].label := wstring#'4';
           #settings.current.kp8.buttons[3].label := wstring#'2';
           #settings.current.kp8.buttons[5].label := wstring#'5';
           #settings.current.kp8.buttons[6].label := wstring#'3';
           #settings.current.kp8.buttons[7].label := wstring#'1';
       END_IF;
   END_REGION

   REGION "CHANGE DETECTION"
       #oldSelState := #settings.current.kp8.btnSelState;
   END_REGION
END_FUNCTION_BLOCK

FUNCTION_BLOCK "Station Details"   // FB22, SCL
{ S7_Optimized_Access := 'TRUE' }
VERSION : 0.1
   VAR_INPUT
      constants : "Constants";
   END_VAR
   VAR_IN_OUT
      settings : "Settings Screen";
      stations : "Stations";
   END_VAR
   VAR
      old : Struct
         nextPress : Bool;
         prevPress : Bool;
         selBtnCount : Int;
         selBtnNumber : Int;
         selStnCount : Int;
         selStnNumber : Int;
      END_STRUCT;
      selStnNumber : Int;
      selBtnNumber : Int;
      newViewReq : Bool;
      instPNEntEnable : "Enable Assignment Pair";
      instAlltEntEnable : "Enable Assignment Pair";
      instCrtEntEnable : "Enable Assignment Pair";
   END_VAR
   VAR_TEMP
      animate : USInt;
      btnCount : Int;
      btnPress : Bool;
      btnSelected : Bool;
      disable : Bool;
      dropZone : WString;
      enable : Bool;
      i : Int;
      line : WString;
      partNumber : WString;
      pBtn : Int;
      selBtnCount : Int;
      selStnCount : Int;
      stnCount : Int;
      stnName : WString;
      stnSelected : Bool;
      timerVal : WString;
   END_VAR
   VAR CONSTANT
      blankString : WString;
   END_VAR
BEGIN
   REGION "POPULATE STATION NAME AND NUMBER"

       REGION "COPY TO LOCAL"
           #selStnCount := #settings.current.stations.selCount;
           #stnCount := #constants.stationCount - 1;
       END_REGION

       REGION "ON CHANGE IN STATION COUNT"
           IF #selStnCount <> #old.selStnCount AND #selStnCount <> 0 THEN

               REGION "FOR EACH STATION"
                   FOR #i := 0 TO #stnCount DO

                       REGION "COPY TO LOCAL"
                           #stnSelected := #stations.current[#i].settings.selected;
                       END_REGION

                       REGION "ON SELECTED STATION"
                           IF #stnSelected THEN

                               #selStnNumber := #i ;
                               EXIT;

                           END_IF;
                       END_REGION

                   END_FOR;
               END_REGION

           END_IF;
       END_REGION

       REGION "CHANGE DETECTION"
           #old.selStnCount := #selStnCount;
       END_REGION

   END_REGION

   REGION "PREVIOUS STATION"

       REGION "COPY TO LOCAL"
           #selStnCount := #settings.current.stations.selCount;
       END_REGION

       REGION "WHILE A STATION HAS BEEN SELECTED"
           IF #selStnCount <> 0 THEN

               REGION "COPY TO LOCAL"
                   #btnPress := #settings.current.viewingStation.previous.actuate;
                   #stnCount := #constants.stationCount - 1;
               END_REGION

               REGION "ON BUTTON PRESS RISING EDGE"
                   IF #btnPress AND NOT #old.prevPress THEN

                       REGION "INITIALIZE INDEX VARIABLE"
                           #i := #selStnNumber - 1;
                       END_REGION

                       REGION "LOW LIMIT ROLL OVER"
                           IF #i < 0 THEN
                               #i := #stnCount;
                           END_IF;
                       END_REGION

                       REGION "COPY TO LOCAL"
                           #stnSelected := #stations.current[#i].settings.selected;
                       END_REGION

                       REGION "FIND NEXT SELECTED STATION"
                           WHILE NOT #stnSelected DO

                               REGION "DECREMENT INDEX"
                                   #i -= 1;
                               END_REGION

                               REGION "EXIT LOOP NO STATION SELECTED"
                                   IF #i < 0 THEN
                                       #i := #stnCount;
                                   END_IF;
                               END_REGION

                               REGION "SAVE WHILE CONDITION"
                                   #stnSelected := #stations.current[#i].settings.selected;
                               END_REGION

                           END_WHILE;
                       END_REGION

                       REGION "SAVE NEW SELECTED STATION NUMBER"
                           #selStnNumber := #i;
                       END_REGION

                   END_IF;
               END_REGION

               REGION "CHANGE DETECTION"
                   #old.prevPress := #btnPress;
               END_REGION

           END_IF;
       END_REGION

   END_REGION

   REGION "NEXT STATION"

       REGION "COPY TO LOCAL"
           #selStnCount := #settings.current.stations.selCount;
       END_REGION

       REGION "WHILE A STATION HAS BEEN SELECTED"
           IF #selStnCount <> 0 THEN

               REGION "COPY TO LOCAL"
                   #btnPress := #settings.current.viewingStation.next.actuate;
                   #stnCount := #constants.stationCount - 1;
               END_REGION

               REGION "ON BUTTON PRESS RISING EDGE"
                   IF #btnPress AND NOT #old.nextPress OR #selStnCount <> #old.selStnCount THEN

                       REGION "INITIALIZE INDEX VARIABLE"
                           #i := #selStnNumber + 1;
                       END_REGION

                       REGION "LOW LIMIT ROLL OVER"
                           IF #i > #stnCount THEN
                               #i := 0;
                           END_IF;
                       END_REGION

                       REGION "COPY TO LOCAL"
                           #stnSelected := #stations.current[#i].settings.selected;
                       END_REGION

                       REGION "FIND NEXT SELECTED STATION"
                           WHILE NOT #stnSelected DO

                               REGION "DECREMENT INDEX"
                                   #i += 1;
                               END_REGION

                               REGION "EXIT LOOP NO STATION SELECTED"
                                   IF #i > #stnCount THEN
                                       #i := 0;
                                   END_IF;
                               END_REGION

                               REGION "SAVE WHILE CONDITION"
                                   #stnSelected := #stations.current[#i].settings.selected;
                               END_REGION

                           END_WHILE;
                       END_REGION

                       REGION "SAVE NEW SELECTED STATION NUMBER"
                           #selStnNumber := #i;
                       END_REGION

                   END_IF;
               END_REGION

               REGION "CHANGE DETECTION"
                   #old.nextPress := #btnPress;
               END_REGION

           END_IF;
       END_REGION


   END_REGION

   REGION "UPDATE STATION NAME"

       REGION "ON CHANGE IN SELECTED STAION NUMBER"
           IF #selStnNumber <> #old.selStnNumber THEN

               REGION "WRITE STATION NAME"
                   #line := #stations.current[#selStnNumber].line;
                   #dropZone := "Strip Sign"(USINT_TO_WSTRING(#stations.current[#selStnNumber].dropZone));
                   #stnName := CONCAT_WSTRING(IN1 := #line,
                                              IN2 := wstring#' ',
                                              IN3 := #dropZone);
                   #settings.current.viewingStation.name := #stnName;
               END_REGION

           END_IF;
       END_REGION



   END_REGION

   REGION "DISPLAY PN AND TIMER VALUES FOR BUTTON"

       REGION "COPY TO LOCAL"
           #selStnCount := #settings.current.stations.selCount;
           #selBtnCount := #settings.current.kp8.selCount;
           #selBtnNumber := #settings.current.kp8.selBtnNumber;
       END_REGION

       REGION "IF A STATION AND BUTTON HAVE BEEN SELECTED"
           IF #selStnCount <> 0 AND #selBtnCount <> 0 THEN

               REGION "ON NEW BUTTON SELECTION"
                   IF #selBtnCount <> #old.selBtnCount OR #selStnCount <> #old.selStnCount THEN

                       REGION "PART NUMBER"
                           #partNumber := #stations.current[#selStnNumber].partNumbers[#selBtnNumber];
                           #settings.current.partNumber.ioField.value := #partNumber;
                       END_REGION

                       REGION "ALLOTTED TIMER"
                           #timerVal := "Real to WString Timer"(#stations.current[#selStnNumber].presetTime.allotted[#selBtnNumber]);
                           #settings.current.alotted.ioField.value := #timerVal;
                       END_REGION

                       REGION "CRITITCAL TIMER"
                           #timerVal := "Real to WString Timer"(#stations.current[#selStnNumber].presetTime.critical[#selBtnNumber]);
                           #settings.current.critical.ioField.value := #timerVal;
                       END_REGION

                   END_IF;
               END_REGION

           END_IF;
       END_REGION

       REGION "ON NO SELECTION"
           IF #selStnCount = 0 OR #selBtnCount = 0 THEN

               REGION "PART NUMBER"
                   #settings.current.partNumber.ioField.value := #blankString;
               END_REGION

               REGION "ALLOTTED TIMER"
                   #settings.current.alotted.ioField.value := #blankString;
               END_REGION

               REGION "CRITITCAL TIMER"
                   #settings.current.critical.ioField.value := #blankString;
               END_REGION

           END_IF;
       END_REGION

   END_REGION

   REGION "LOAD BUTTON DETAILS"

       REGION "COPY TO LOCAL"
           #selStnCount := #settings.current.stations.selCount;
           #btnCount := #constants.buttonCount - 3;
       END_REGION

       REGION "ON SELECTED STATIONS"
           IF #selStnCount >= 1 THEN

               REGION "FOR EACH BUTTON"
                   FOR #i := 0 TO #btnCount DO

                       REGION "CALCULATE BUTTON POINTER"
                           IF #i MOD 2 = 0 THEN
                               #pBtn := 7 - #i / 2;
                           END_IF;
                           IF #i MOD 2 <> 0 THEN
                               #pBtn := 3 - #i / 2;
                           END_IF;
                       END_REGION

                       REGION "BUTTON LABEL"
                           #settings.current.viewingStation.btns[#i].label.value := "Strip Sign"(INT_TO_WSTRING(#i + 1));
                       END_REGION

                       REGION "ALLOTTED TIME"
                           #timerVal := "Real to WString Timer"(#stations.current[#selStnNumber].presetTime.allotted[#pBtn]);
                           #settings.current.viewingStation.btns[#i].alloted.value := #timerVal;
                       END_REGION

                       REGION "CRITICAL TIME"
                           #timerVal := "Real to WString Timer"(#stations.current[#selStnNumber].presetTime.critical[#pBtn]);
                           #settings.current.viewingStation.btns[#i].critical.value := #timerVal;
                       END_REGION

                       REGION "PART NUMBER"
                           #partNumber := #stations.current[#selStnNumber].partNumbers[#pBtn];
                           #settings.current.viewingStation.btns[#i].partNumber.value := #partNumber;
                       END_REGION

                   END_FOR;
               END_REGION

           END_IF;
       END_REGION

   END_REGION

   REGION "ANIMATIONS"

       REGION "COPY TO LOCAL"
           #selStnCount := #settings.current.stations.selCount;
       END_REGION

       REGION "PN AND TIMERS"

           REGION "ENABLE/DISABLE FOR PN AND TIMERS"

               REGION "SET DISABLE"
                   IF #selStnCount = 0 OR #selBtnCount = 0 THEN
                       #disable := TRUE;
                       #enable := FALSE;
                   END_IF;
               END_REGION

               REGION "SET ENABLE"
                   IF #selStnCount <> 0 AND #selBtnCount <> 0 THEN
                       #disable := FALSE;
                       #enable := TRUE;
                   END_IF;
               END_REGION

           END_REGION

           REGION "PN ANIMATION FUNCTIONS"
               #animate := #settings.current.partNumber.assign.animate;
               #instPNEntEnable(constants := #constants,
                                disable := #disable,
                                enable := #enable,
                                value := #settings.current.partNumber.ioField.value,
                                assignAnimate := #animate,
                                ioFieldAnimate := #settings.current.partNumber.ioField.animate);
               #animate := "Animate Bool"(colorTrue := #constants.colorLib.BgLGr,
                                          colorFalse := #animate,
                                          evalSignal := #settings.current.partNumber.assign.actuate);
               #settings.current.partNumber.assign.animate := #animate;
           END_REGION

           REGION "ALLOTTED TIME ANIMATION FUNCTIONS"
               #animate := #settings.current.alotted.assign.animate;
               #instAlltEntEnable(constants := #constants,
                                  disable := #disable,
                                  enable := #enable,
                                  value := #settings.current.alotted.ioField.value,
                                  assignAnimate := #animate,
                                  ioFieldAnimate := #settings.current.alotted.ioField.animate);
               #animate := "Animate Bool"(colorTrue := #constants.colorLib.BgLGr,
                                          colorFalse := #animate,
                                          evalSignal := #settings.current.alotted.assign.actuate);
               #settings.current.alotted.assign.animate := #animate;
           END_REGION

           REGION "CRITICAL TIME ANIMATION FUNCTIONS"
               #animate := #settings.current.critical.assign.animate;
               #instCrtEntEnable(constants := #constants,
                                 disable := #disable,
                                 enable := #enable,
                                 value := #settings.current.critical.ioField.value,
                                 assignAnimate := #animate,
                                 ioFieldAnimate := #settings.current.critical.ioField.animate);
               #animate := "Animate Bool"(colorTrue := #constants.colorLib.BgLGr,
                                          colorFalse := #animate,
                                          evalSignal := #settings.current.critical.assign.actuate);
               #settings.current.critical.assign.animate := #animate;
           END_REGION

       END_REGION

       REGION "PREVIOUS STATION"
           #animate := "Animate Bool"(colorTrue := #constants.colorLib.BgLGr,
                                      colorFalse := #constants.colorLib.BgGray,
                                      evalSignal := #settings.current.viewingStation.previous.actuate);
           #settings.current.viewingStation.previous.animate := #animate;
       END_REGION

       REGION "NEXT STATION"
           #animate := "Animate Bool"(colorTrue := #constants.colorLib.BgLGr,
                                      colorFalse := #constants.colorLib.BgGray,
                                      evalSignal := #settings.current.viewingStation.next.actuate);
           #settings.current.viewingStation.next.animate := #animate;
       END_REGION

       REGION "ENABLE/DISABLE LINE DISPLAY"

           REGION "ENABLE"
               IF #selStnCount = 1 THEN
                   #settings.current.viewingStation.lineData.animate.bg := #constants.colorLib.BgGray;
                   #settings.current.viewingStation.lineData.animate.ioField := #constants.colorLib.BgWh;
               END_IF;
           END_REGION

           REGION "DISABLE"
               IF #selStnCount <> 1 THEN
                   #settings.current.viewingStation.lineData.animate.bg := #constants.colorLib.invisible;
                   #settings.current.viewingStation.lineData.animate.ioField := #constants.colorLib.invisible;
               END_IF;
           END_REGION

       END_REGION

       REGION "ENABLE/DISABLE DROPZONE"

           REGION "ENABLE"
               IF #selStnCount = 1 THEN
                   #settings.current.viewingStation.dzData.animate.bg := #constants.colorLib.BgGray;
                   #settings.current.viewingStation.dzData.animate.ioField := #constants.colorLib.BgWh;
               END_IF;
           END_REGION

           REGION "DISABLE"
               IF #selStnCount <> 1 THEN
                   #settings.current.viewingStation.dzData.animate.bg := #constants.colorLib.invisible;
                   #settings.current.viewingStation.dzData.animate.ioField := #constants.colorLib.invisible;
               END_IF;
           END_REGION

       END_REGION

       REGION "ENABLE/DISABLE BUTTON DETAILS"

           REGION "COPY TO LOCAL"
               #btnCount := #constants.buttonCount - 3;
           END_REGION

           REGION "ENABLE"
               IF #selStnCount >= 1 THEN

                   REGION "SHOW BUTTON DETAILS"
                       #animate := #constants.colorLib.BgGray;
                   END_REGION

               END_IF;
           END_REGION

           REGION "DISABLE"
               IF #selStnCount = 0 THEN

                   REGION "HIDE BUTTON DETAILS"
                       #animate := #constants.colorLib.invisible;
                   END_REGION

               END_IF;
           END_REGION

           REGION "APPLY ANIMATION"
               FOR #i := 0 TO #btnCount DO
                   #settings.current.viewingStation.btns[#i].label.animate := #animate;
                   #settings.current.viewingStation.btns[#i].alloted.animate := #animate;
                   #settings.current.viewingStation.btns[#i].critical.animate := #animate;
                   #settings.current.viewingStation.btns[#i].partNumber.animate := #animate;
               END_FOR;

           END_REGION 
       END_REGION

   END_REGION

   REGION "CHANGE DETECTION"
       #old.selStnNumber := #selStnNumber;
       #old.selBtnNumber := #selBtnNumber;
       #old.selBtnCount := #selBtnCount;
       #old.selStnCount := #selStnCount;
   END_REGION
END_FUNCTION_BLOCK

FUNCTION_BLOCK "Enable Assignment Pair"   // FB23, SCL
{ S7_Optimized_Access := 'TRUE' }
VERSION : 0.1
   VAR_INPUT
      constants : "Constants";
      disable : Bool;
      enable : Bool;
   END_VAR
   VAR_IN_OUT
      value : WString;
      assignAnimate : USInt;
      ioFieldAnimate : USInt;
   END_VAR
   VAR
      old : Struct
         disabled : Bool;
         enabled : Bool;
      END_STRUCT;
   END_VAR
BEGIN
   REGION "DISABLED"    
       IF #disable THEN
           #value := wstring#'';
           #assignAnimate := #constants.colorLib.disabled;
           #ioFieldAnimate := #constants.colorLib.disabled;
       END_IF;
   END_REGION

   REGION "ENABLED"
           IF #enable THEN
               #assignAnimate := #constants.colorLib.BgGray;
               #ioFieldAnimate := #constants.colorLib.BgWh;
           END_IF;
   END_REGION
END_FUNCTION_BLOCK

FUNCTION_BLOCK "KP8 Driver"   // FB101, SCL
{ S7_Optimized_Access := 'FALSE' }
VERSION : 0.1
   VAR_INPUT
      btnIn : Byte;   // byte that contains input data from kp8 buttons
      hardInit : Bool;   // initializes function. can be used for reset
      softInit : Bool;
      btn0Activate : Bool;   // true for on, false for off
      btn0Mode : Bool;   // true for maintained, false for momentary
      btn0Group : Int;
      btn0Flash : Bool;
      btn0ColorOn1 : String[10];   // enter: red OR green OR blue OR yellow OR white OR off
      btn0ColorOn2 : String[10];
      btn0ColorOff : String[10];   // enter: red OR green OR blue OR yellow OR white OR off
      btn1Activate : Bool;   // true for on, false for off
      btn1Mode : Bool;   // true for maintained, false for momentary
      btn1Group : Int;
      btn1Flash : Bool;
      btn1ColorOn1 : String[10];   // enter: red OR green OR blue OR yellow OR white OR off
      btn1ColorOn2 : String[10];
      btn1ColorOff : String[10];   // enter: red OR green OR blue OR yellow OR white OR off
      btn2Activate : Bool;   // true for on, false for off
      btn2Mode : Bool;   // true for maintained, false for momentary
      btn2Group : Int;
      btn2Flash : Bool;
      btn2ColorOn1 : String[10] := '';   // enter: red OR green OR blue OR yellow OR white OR off
      btn2ColorOn2 : String[10];
      btn2ColorOff : String[10];   // enter: red OR green OR blue OR yellow OR white OR off
      btn3Activate : Bool;   // true for on, false for off
      btn3Mode : Bool;   // true for maintained, false for momentary
      btn3Group : Int;
      btn3Flash : Bool;
      btn3ColorOn1 : String[10];   // enter: red OR green OR blue OR yellow OR white OR off
      btn3ColorOn2 : String[10];
      btn3ColorOff : String[10];   // enter: red OR green OR blue OR yellow OR white OR off
      btn4Activate : Bool;   // true for on, false for off
      btn4Mode : Bool;   // true for maintained, false for momentary
      btn4Group : Int;
      btn4Flash : Bool;
      btn4ColorOn1 : String[10];   // enter: red OR green OR blue OR yellow OR white OR off
      btn4ColorOn2 : String[10];
      btn4ColorOff : String[10];   // enter: red OR green OR blue OR yellow OR white OR off
      btn5Activate : Bool;   // true for on, false for off
      btn5Mode : Bool;   // true for maintained, false for momentary
      btn5Group : Int;
      btn5Flash : Bool;
      btn5ColorOn1 : String[10];   // enter: red OR green OR blue OR yellow OR white OR off
      btn5ColorOn2 : String[10];
      btn5ColorOff : String[10];   // enter: red OR green OR blue OR yellow OR white OR off
      btn6Activate : Bool;   // true for on, false for off
      btn6Mode : Bool;   // true for maintained, false for momentary
      btn6Group : Int;
      btn6Flash : Bool;
      btn6ColorOn1 : String[10];   // enter: red OR green OR blue OR yellow OR white OR off
      btn6ColorOn2 : String[10];
      btn6ColorOff : String[10];   // enter: red OR green OR blue OR yellow OR white OR off
      btn7Activate : Bool;   // true for on, false for off
      btn7Mode : Bool;   // true for maintained, false for momentary
      btn7Group : Int;
      btn7Flash : Bool;
      btn7ColorOn1 : String[10];   // enter: red OR green OR blue OR yellow OR white OR off
      btn7ColorOn2 : String[10];
      btn7ColorOff : String[10];   // enter: red OR green OR blue OR yellow OR white OR off
   END_VAR
   VAR_OUTPUT
      btnStatesOut : Array[0..7] of Bool;   // the output array represents the state of button presses
      btnColorsOut : DWord;
   END_VAR
   VAR
      mask : Byte;
      btnInInt : Byte;
      btnEval : Byte;
      i1 : Int;
      i2 : Int;
      btnInArrayNew : Array[0..7] of Bool;
      btnInArrayOld : Array[0..7] of Bool;
      btnStateArrayInt : Array[0..7] of Bool;
      btnActivateInt : Array[0..7] of Bool;
      btnModeInt : Array[0..7] of Bool;
      btnFlashInt : Array[0..7] of Bool;
      btnGroup : Array[0..7] of Int;
      btnClrMskOn1Int : Array[0..7] of DWord;
      btnClrMskOn2Int : Array[0..7] of DWord;
      btnClrMskOffInt : Array[0..7] of DWord;
      btnClrOn1Int : Array[0..7] of String[10];
      btnClrOn2Int : Array[0..7] of String[10];
      btnClrOffInt : Array[0..7] of String[10];
   END_VAR
   VAR CONSTANT
      btnMskRed : DWord := dw#16#0100_0000;
      btnMskGreen : DWord := dw#16#0001_0000;
      btnMskBlue : DWord := dw#16#000_0100;
      btnMskYellow : DWord := dw#16#0101_0000;
      btnMskWhite : DWord := dw#16#0101_0100;
      btnMskBlack : DWord := dw#16#FEFE_FEFF;
      initBtnColors : DWord := dw#16#0000_0000;
   END_VAR
BEGIN
   REGION "ALL INITS"
       IF #hardInit OR #softInit THEN

           REGION "CLEAR OUTPUT COLORS"
               #btnColorsOut := #initBtnColors;
           END_REGION

           REGION "TRANSFER PARAMETERS TO INTERNAL ARRAYS"

               REGION "BUTTON 0"
                   #btnActivateInt[0] := #btn0Activate;
                   #btnModeInt[0] := #btn0Mode;
                   #btnGroup[0] := #btn0Group;
                   #btnClrOn1Int[0] := #btn0ColorOn1;
                   #btnClrOn2Int[0] := #btn0ColorOn2;
                   #btnClrOffInt[0] := #btn0ColorOff;
               END_REGION

               REGION "BUTTON 1"
                   #btnActivateInt[1] := #btn1Activate;
                   #btnModeInt[1] := #btn1Mode;
                   #btnGroup[1] := #btn1Group;
                   #btnClrOn1Int[1] := #btn1ColorOn1;
                   #btnClrOn2Int[1] := #btn1ColorOn2;
                   #btnClrOffInt[1] := #btn1ColorOff;
               END_REGION

               REGION "BUTTON 2"
                   #btnActivateInt[2] := #btn2Activate;
                   #btnModeInt[2] := #btn2Mode;
                   #btnGroup[2] := #btn2Group;
                   #btnClrOn1Int[2] := #btn2ColorOn1;
                   #btnClrOn2Int[2] := #btn2ColorOn2;
                   #btnClrOffInt[2] := #btn2ColorOff;
               END_REGION

               REGION "BUTTON 3"
                   #btnActivateInt[3] := #btn3Activate;
                   #btnModeInt[3] := #btn3Mode;
                   #btnGroup[3] := #btn3Group;
                   #btnClrOn1Int[3] := #btn3ColorOn1;
                   #btnClrOn2Int[3] := #btn3ColorOn2;
                   #btnClrOffInt[3] := #btn3ColorOff;
               END_REGION

               REGION "BUTTON 4"
                   #btnActivateInt[4] := #btn4Activate;
                   #btnModeInt[4] := #btn4Mode;
                   #btnGroup[4] := #btn4Group;
                   #btnClrOn1Int[4] := #btn4ColorOn1;
                   #btnClrOn2Int[4] := #btn4ColorOn2;
                   #btnClrOffInt[4] := #btn4ColorOff;
               END_REGION

               REGION "BUTTON 5"
                   #btnActivateInt[5] := #btn5Activate;
                   #btnModeInt[5] := #btn5Mode;
                   #btnGroup[5] := #btn5Group;
                   #btnClrOn1Int[5] := #btn5ColorOn1;
                   #btnClrOn2Int[5] := #btn5ColorOn2;
                   #btnClrOffInt[5] := #btn5ColorOff;
               END_REGION

               REGION "BUTTON 6"
                   #btnActivateInt[6] := #btn6Activate;
                   #btnModeInt[6] := #btn6Mode;
                   #btnGroup[6] := #btn6Group;
                   #btnClrOn1Int[6] := #btn6ColorOn1;
                   #btnClrOn2Int[6] := #btn6ColorOn2;
                   #btnClrOffInt[6] := #btn6ColorOff;
               END_REGION

               REGION "BUTTON 7"
                   #btnActivateInt[7] := #btn7Activate;
                   #btnModeInt[7] := #btn7Mode;
                   #btnGroup[7] := #btn7Group;
                   #btnClrOn1Int[7] := #btn7ColorOn1;
                   #btnClrOn2Int[7] := #btn7ColorOn2;
                   #btnClrOffInt[7] := #btn7ColorOff;
               END_REGION

           END_REGION

           REGION "RECOLOR BUTTON MASKS"
               FOR #i1 := 0 TO 7 DO

                   REGION "ON COLOR 1"
                       IF (#btnClrOn1Int[#i1] = 'red') THEN
                           #btnClrMskOn1Int[#i1] := SHL(IN := #btnMskRed, N := #i1);
                       ELSIF (#btnClrOn1Int[#i1] = 'green') THEN
                           #btnClrMskOn1Int[#i1] := SHL(IN := #btnMskGreen, N := #i1);
                       ELSIF (#btnClrOn1Int[#i1] = 'blue') THEN
                           #btnClrMskOn1Int[#i1] := SHL(IN := #btnMskBlue, N := #i1);
                       ELSIF (#btnClrOn1Int[#i1] = 'yellow') THEN
                           #btnClrMskOn1Int[#i1] := SHL(IN := #btnMskYellow, N := #i1);
                       ELSIF (#btnClrOn1Int[#i1] = 'white') THEN
                           #btnClrMskOn1Int[#i1] := SHL(IN := #btnMskWhite, N := #i1);
                       ELSIF (#btnClrOn1Int[#i1] = 'off') THEN
                           #btnClrMskOn1Int[#i1] := 0;
                       END_IF;
                   END_REGION

                   REGION "ON COLOR 2"
                       IF (#btnClrOn2Int[#i1] = 'red') THEN
                           #btnClrMskOn2Int[#i1] := SHL(IN := #btnMskRed, N := #i1);
                       ELSIF (#btnClrOn2Int[#i1] = 'green') THEN
                           #btnClrMskOn2Int[#i1] := SHL(IN := #btnMskGreen, N := #i1);
                       ELSIF (#btnClrOn2Int[#i1] = 'blue') THEN
                           #btnClrMskOn2Int[#i1] := SHL(IN := #btnMskBlue, N := #i1);
                       ELSIF (#btnClrOn2Int[#i1] = 'yellow') THEN
                           #btnClrMskOn2Int[#i1] := SHL(IN := #btnMskYellow, N := #i1);
                       ELSIF (#btnClrOn2Int[#i1] = 'white') THEN
                           #btnClrMskOn2Int[#i1] := SHL(IN := #btnMskWhite, N := #i1);
                       ELSIF (#btnClrOn2Int[#i1] = 'off') THEN
                           #btnClrMskOn2Int[#i1] := 0;
                       END_IF;
                   END_REGION

                   REGION "OFF COLOR"
                       IF (#btnClrOffInt[#i1] = 'red') THEN
                           #btnClrMskOffInt[#i1] := SHL(IN := #btnMskRed, N := #i1);
                       ELSIF (#btnClrOffInt[#i1] = 'green') THEN
                           #btnClrMskOffInt[#i1] := SHL(IN := #btnMskGreen, N := #i1);
                       ELSIF (#btnClrOffInt[#i1] = 'blue') THEN
                           #btnClrMskOffInt[#i1] := SHL(IN := #btnMskBlue, N := #i1);
                       ELSIF (#btnClrOffInt[#i1] = 'yellow') THEN
                           #btnClrMskOffInt[#i1] := SHL(IN := #btnMskYellow, N := #i1);
                       ELSIF (#btnClrOffInt[#i1] = 'white') THEN
                           #btnClrMskOffInt[#i1] := SHL(IN := #btnMskWhite, N := #i1);
                       ELSIF (#btnClrOffInt[#i1] = 'off') THEN
                           #btnClrMskOffInt[#i1] := 0;
                       END_IF;
                   END_REGION

               END_FOR;
           END_REGION

       END_IF;
   END_REGION

   REGION "HART INIT"
       IF #hardInit THEN
           FOR #i1 := 0 TO 7 DO
               #btnStateArrayInt[#i1] := FALSE;
           END_FOR;
       END_IF;
   END_REGION


   REGION "TRANFER PARAMETERS TO ARRAYS"
       // raw pb data
       #btnInInt := #btnIn;
       // flashing modes
       #btnFlashInt[0] := #btn0Flash;
       #btnFlashInt[1] := #btn1Flash;
       #btnFlashInt[2] := #btn2Flash;
       #btnFlashInt[3] := #btn3Flash;
       #btnFlashInt[4] := #btn4Flash;
       #btnFlashInt[5] := #btn5Flash;
       #btnFlashInt[6] := #btn6Flash;
       #btnFlashInt[7] := #btn7Flash;
   END_REGION

   REGION "EVALUATE BUTTONS"
       FOR #i1 := 0 TO 7 DO

           REGION "TRANSFER BUTTON PRESSES TO ARRAY"
               #btnEval := SHR(IN := #btnInInt, N := #i1);
               #btnInArrayNew[#i1] := #btnEval.%X0;
               #btnEval := b#16#0;
           END_REGION

           REGION "SET BUTTON STATE"

               REGION "BUTTON ACTIVE"
                   IF #btnActivateInt[#i1] THEN

                       REGION "MAINTAINED"
                           IF #btnModeInt[#i1] THEN

                               REGION "RISING EDGE OF PRESS"
                                   IF #btnInArrayNew[#i1] AND NOT #btnInArrayOld[#i1] THEN

                                       REGION "CHECK FOR GROUP MEMBERSHIP"
                                           FOR #i2 := 0 TO 7 DO

                                               REGION "NOT IN NULL GROUP"
                                                   IF (#btnGroup[#i2] <> 0) THEN

                                                       REGION "SKIP SELF"
                                                           IF (#i2 <> #i1) THEN

                                                               REGION "GROUPS MATCH"
                                                                   IF #btnGroup[#i1] = #btnGroup[#i2] THEN
                                                                       REGION "DEACTIVATE OTHER GROUP MEMBERS"
                                                                           #btnStateArrayInt[#i2] := FALSE;
                                                                       END_REGION

                                                                   END_IF;
                                                               END_REGION

                                                           END_IF;
                                                       END_REGION

                                                   END_IF;
                                               END_REGION

                                           END_FOR;
                                       END_REGION

                                       REGION "TOGGLE STATE"
                                           #btnStateArrayInt[#i1] := NOT #btnStateArrayInt[#i1];
                                       END_REGION

                                   END_IF;
                               END_REGION

                           END_IF;
                       END_REGION

                       REGION "MOMENTARY"
                           IF NOT #btnModeInt[#i1] THEN
                               #btnStateArrayInt[#i1] := #btnInArrayNew[#i1];
                           END_IF;
                       END_REGION

                   END_IF;
               END_REGION

               REGION "BUTTON INACTIVE"
                   IF NOT #btnActivateInt[#i1] THEN
                       #btnStateArrayInt[#i1] := FALSE;
                   END_IF;
               END_REGION

           END_REGION

           REGION "ANIMATE BUTTONS"

               REGION "BUTTON ON FLASH BIT OFF"
                   IF #btnStateArrayInt[#i1] AND NOT #btnFlashInt[#i1] THEN
                       #btnColorsOut := #btnColorsOut AND ROL(IN := #btnMskBlack, N := #i1);
                       #btnColorsOut := #btnColorsOut OR #btnClrMskOn1Int[#i1];
                   END_IF;
               END_REGION

               REGION "BUTTON ON FLASH BIT ON"
                   IF #btnStateArrayInt[#i1] AND #btnFlashInt[#i1] THEN
                       #btnColorsOut := #btnColorsOut AND ROL(IN := #btnMskBlack, N := #i1);
                       #btnColorsOut := #btnColorsOut OR #btnClrMskOn2Int[#i1];
                   END_IF;
               END_REGION

               REGION "BUTTON OFF"
                   IF NOT #btnStateArrayInt[#i1] THEN
                       #btnColorsOut := #btnColorsOut AND ROL(IN := #btnMskBlack, N := #i1);
                       #btnColorsOut := #btnColorsOut OR #btnClrMskOffInt[#i1];
                   END_IF;
               END_REGION

           END_REGION

       END_FOR;
   END_REGION

   REGION "CHANGE DETECTION"
       #btnInArrayOld := #btnInArrayNew;
   END_REGION

   REGION "OUTPUT"
       #btnStatesOut := #btnStateArrayInt;
   END_REGION
END_FUNCTION_BLOCK

FUNCTION "Physical to Global" : Void   // FC1, LAD
{ S7_Optimized_Access := 'TRUE' }
VERSION : 0.1
   VAR_INPUT
      constants : "Constants";
   END_VAR
   VAR_IN_OUT
      stations : "Stations";
   END_VAR
   VAR_TEMP
      i : Int;
      kp8In : DWord;
      stnCount : Int;
   END_VAR
   VAR CONSTANT
      "VOLVO 16 1" : Int := 0;
      "VOLVO 16 2" : Int := 1;
      "VOLVO 16 3" : Int := 2;
      "VOLVO 16 4" : Int := 3;
      "VOLVO 16 5" : Int := 4;
      "VOLVO 16 6" : Int := 5;
      "VOLVO 16 7" : Int := 6;
      "VOLVO 16 8" : Int := 7;
      "VOLVO 16 9" : Int := 8;
      "VOLVO 16 10" : Int := 9;
      "VOLVO 16 11" : Int := 10;
      "CHM 01" : Int := 11;
      "CHM 02" : Int := 12;
      "CHM 03" : Int := 13;
      "CHM 04" : Int := 14;
      "CHM 05" : Int := 15;
      "CDO 01" : Int := 16;
      "CDO 02" : Int := 17;
      "CDO 03" : Int := 18;
      "BFL 01" : Int := 19;
      "BFL 02" : Int := 20;
      "BFL 03" : Int := 21;
      "LGS 01" : Int := 22;
      "LGS 02" : Int := 23;
   END_VAR
BEGIN

REGION Network 1
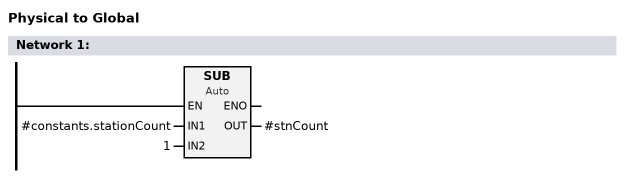
   RUNG wire#powerrail
      Sub(in1 := #constants.stationCount, in2 := 1, out => #stnCount)
   END_RUNG
   // the same network as SCL:
   #stnCount := #constants.stationCount - 1;
END_REGION

REGION Network 2 (SCL): MAIN LOOP
   FOR #i := 0 TO #stnCount DO

       CASE #i OF
           #"VOLVO 16 1":
               #kp8In := "VOLVO 16 01 KP8 In";
           #"VOLVO 16 2":
               #kp8In := "VOLVO 16 02 KP8 In";
           #"VOLVO 16 3":
               #kp8In := "VOLVO 16 03 KP8 In";
           #"VOLVO 16 4":
               #kp8In := "VOLVO 16 04 KP8 In";
           #"VOLVO 16 5":
               #kp8In := "VOLVO 16 05 KP8 In";
           #"VOLVO 16 6":
               #kp8In := "VOLVO 16 06 KP8 In";
           #"VOLVO 16 7":
               #kp8In := "VOLVO 16 07 KP8 In";
           #"VOLVO 16 8":
               #kp8In := "VOLVO 16 08 KP8 In";
           #"VOLVO 16 9":
               #kp8In := "VOLVO 16 09 KP8 In";
           #"VOLVO 16 10":
               #kp8In := "VOLVO 16 10 KP8 In";
           #"VOLVO 16 11":
               #kp8In := "VOLVO 16 11 KP8 In";
           #"CHM 01":
               #kp8In := "CHM 01 KP8 In";
           #"CHM 02":
               #kp8In := "CHM 02 KP8 In";
           #"CHM 03":
               #kp8In := "CHM 03 KP8 In";
           #"CHM 04":
               #kp8In := "CHM 04 KP8 In";
           #"CHM 05":
               #kp8In := "CHM 05 KP8 In";
           #"CDO 01":
               #kp8In := "CDO 01 KP8 In";
           #"CDO 02":
               #kp8In := "CDO 02 KP8 In";
           #"CDO 03":
               #kp8In := "CDO 03 KP8 In";
           #"BFL 01":
               #kp8In := "BFL 01 KP8 In";
           #"BFL 02":
               #kp8In := "BFL 02 KP8 In";
           #"BFL 03":
               #kp8In := "BFL 03 KP8 In";
           #"LGS 01":
               #kp8In := "LGS 01 KP8 In";
           #"LGS 02":
               #kp8In := "LGS 02 KP8 In";

       END_CASE;

       #stations.current[#i].kp8In := #kp8In.%B3;

   END_FOR;
END_REGION
END_FUNCTION

FUNCTION "Time to WString" : WString   // FC2, SCL
{ S7_Optimized_Access := 'TRUE' }
VERSION : 0.1
   VAR_INPUT
      "Time" : Time;
   END_VAR
   VAR_TEMP
      "Time as DInt" : DInt;
      "Hours 10s Place" : DInt;
      "Hours 1s Place" : DInt;
      "Minutes 10s Place" : DInt;
      "Minutes 1s Place" : DInt;
      "Seconds 10s Place" : DInt;
      "Seconds 1s Place" : DInt;
      "Time Elements" : Array[0..4] of WString;
      Length : Int;
      "String Box" : WString;
      "DInt Box" : DInt;
   END_VAR
   VAR CONSTANT
      "Milliseconds per 10 Hours" : DInt := 36000000;
      "Milliseconds per Hour" : DInt := 3600000;
      "Milliseconds per 10 Minutes" : DInt := 600000;
      "Milliseconds per Minute" : DInt := 60000;
      "Milliseconds per 10 Seconds" : DInt := 10000;
      "Milliseconds per Second" : DInt := 1000;
   END_VAR
BEGIN
   REGION GET INPUT
       #"Time as DInt" := #Time;
   END_REGION

   REGION CONVERT TIME INTO INDIVIDUAL PLACE VALUES
       #"Minutes 10s Place" := #"Time as DInt" / #"Milliseconds per 10 Minutes";
       #"Minutes 1s Place" := (#"Time as DInt" / #"Milliseconds per Minute") MOD 10;
       #"Seconds 10s Place" := (#"Time as DInt" MOD #"Milliseconds per Minute") / #"Milliseconds per 10 Seconds";
       #"Seconds 1s Place" := (#"Time as DInt" / #"Milliseconds per Second") MOD 10;
   END_REGION

   REGION "ADD SIGN"
       #"Time Elements"[0] := wstring#'';
       IF #"Minutes 10s Place" < 0 OR
           #"Minutes 1s Place" < 0 OR
           #"Seconds 10s Place" < 0 OR
           #"Seconds 1s Place" < 0 THEN
            #"Time Elements"[0] := wstring#'-';
       END_IF;
   END_REGION

   REGION CONVERT PLACE VALUES INTO COMPONENT STRINGS
       // MINUTES
       #"DInt Box" := #"Minutes 10s Place" * 10 + #"Minutes 1s Place";
       #"String Box" := DINT_TO_WSTRING(IN := #"DInt Box");
       #"String Box" := "Strip Sign"("WString":=#"String Box");
       #"String Box" := "Add Leading"("Leading Character" := WCHAR#'0',
                                      "Desired Length" := 2,
                                      "String" := #"String Box");
       #"Time Elements"[1] := #"String Box";
       // COLON
       #"Time Elements"[2] := WSTRING#':';
       // SECONDS
       #"DInt Box" := #"Seconds 10s Place" * 10 + #"Seconds 1s Place";
       #"String Box" := DINT_TO_WSTRING(IN := #"DInt Box");
       #"String Box" := "Strip Sign"("WString":=#"String Box");
       #"String Box" := "Add Leading"("Leading Character" := WCHAR#'0',
                                      "Desired Length" := 2,
                                      "String" := #"String Box");
       #"Time Elements"[3] := #"String Box";
   END_REGION


   REGION RETURN VALUE
       #"Time to WString" := CONCAT_WSTRING(IN1 := #"Time Elements"[0],
                                            IN2 := #"Time Elements"[1],
                                            IN3 := #"Time Elements"[2],
                                            IN4 := #"Time Elements"[3]);
   END_REGION
END_FUNCTION

FUNCTION "Strip Sign" : WString   // FC3, SCL
{ S7_Optimized_Access := 'TRUE' }
VERSION : 0.1
   VAR_INPUT
      WString : WString;
   END_VAR
   VAR_TEMP
      Length : Int;
      "String Box" : WString;
      "Test Character" : WString;
   END_VAR
   VAR CONSTANT
      "+" : WChar := WCHAR#'+';
      "-" : WChar := WCHAR#'-';
   END_VAR
BEGIN
   #"String Box" := #WString;
   #"Test Character" := LEFT_WSTRING(IN := #"String Box",
                                     L := 1);
   IF #"Test Character" = #"+" OR #"Test Character" = #"-" THEN
       #Length := LEN(#"String Box");
       #"String Box" := RIGHT_WSTRING(IN := #"String Box", L := #Length - 1);

   END_IF;
   #"Strip Sign" := #"String Box";
END_FUNCTION

FUNCTION "Add Leading" : WString   // FC4, SCL
{ S7_Optimized_Access := 'TRUE' }
VERSION : 0.1
   VAR_INPUT
      "Leading Character" : WChar;
      "Desired Length" : USInt;
      "String" : WString;
   END_VAR
   VAR_TEMP
      Length : Int;
      "String Box" : WString;
      Constant : WString;
   END_VAR
BEGIN
   #"String Box" := #String;
   #Length := LEN(#"String Box");

   WHILE #Length < #"Desired Length" DO
       #"String Box" := CONCAT_WSTRING(IN1 := #"Leading Character",
                                       IN2 := #"String Box");
       #Length := LEN(#"String Box");
   END_WHILE;

   #"Add Leading" := #"String Box";
END_FUNCTION

FUNCTION "Global to Physical" : Void   // FC5, LAD
{ S7_Optimized_Access := 'TRUE' }
VERSION : 0.1
   VAR_INPUT
      constants : "Constants";
   END_VAR
   VAR_IN_OUT
      stations : "Stations";
   END_VAR
   VAR_TEMP
      i : Int;
      j : Int;
      IO : DWord;
      "KP8 In" : DWord;
      "KP8 Out" : DWord;
      Card : Int;
      stnCount : Int;
   END_VAR
   VAR CONSTANT
      "VOLVO 16 01" : Int := 0;
      "VOLVO 16 02" : Int := 1;
      "VOLVO 16 03" : Int := 2;
      "VOLVO 16 04" : Int := 3;
      "VOLVO 16 05" : Int := 4;
      "VOLVO 16 06" : Int := 5;
      "VOLVO 16 07" : Int := 6;
      "VOLVO 16 08" : Int := 7;
      "VOLVO 16 09" : Int := 8;
      "VOLVO 16 10" : Int := 9;
      "VOLVO 16 11" : Int := 10;
      "CHM 01" : Int := 11;
      "CHM 02" : Int := 12;
      "CHM 03" : Int := 13;
      "CHM 04" : Int := 14;
      "CHM 05" : Int := 15;
      "CDO 01" : Int := 16;
      "CDO 02" : Int := 17;
      "CDO 03" : Int := 18;
      "BFL 01" : Int := 19;
      "BFL 02" : Int := 20;
      "BFL 03" : Int := 21;
      "LGS 01" : Int := 22;
      "LGS 02" : Int := 23;
   END_VAR
BEGIN

REGION Network 1: ARRAY LIMIT FOR STATION COUNT
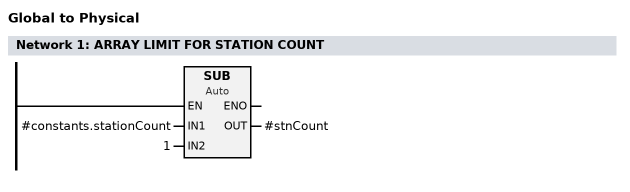
   RUNG wire#powerrail
      Sub(in1 := #constants.stationCount, in2 := 1, out => #stnCount)
   END_RUNG
   // the same network as SCL:
   #stnCount := #constants.stationCount - 1;
END_REGION

REGION Network 2 (SCL): MAIN LOOP
   FOR #i := 0 TO #stnCount DO

       #IO := #stations.current[#i].stackLightOut;
       #"KP8 Out" := #stations.current[#i].kp8Out;

       CASE #i OF
           #"VOLVO 16 01":
               "VOLVO 16 01 IO" := #IO;
               "VOLVO 16 01 KP8 Out" := #"KP8 Out";
           #"VOLVO 16 02":
               "VOLVO 16 02 IO" := #IO;
               "VOLVO 16 02 KP8 Out" := #"KP8 Out";
           #"VOLVO 16 03":
               "VOLVO 16 03 IO" := #IO;
               "VOLVO 16 03 KP8 Out" := #"KP8 Out";
           #"VOLVO 16 04":
               "VOLVO 16 04 IO" := #IO;
               "VOLVO 16 04 KP8 Out" := #"KP8 Out";
           #"VOLVO 16 05":
               "VOLVO 16 05 IO" := #IO;
               "VOLVO 16 05 KP8 Out" := #"KP8 Out";
           #"VOLVO 16 06":
               "VOLVO 16 06 IO" := #IO;
               "VOLVO 16 06 KP8 Out" := #"KP8 Out";
           #"VOLVO 16 07":
               "VOLVO 16 07 IO" := #IO;
               "VOLVO 16 07 KP8 Out" := #"KP8 Out";
           #"VOLVO 16 08":
               "VOLVO 16 08 IO" := #IO;
               "VOLVO 16 08 KP8 Out" := #"KP8 Out";
           #"VOLVO 16 09":
               "VOLVO 16 09 IO" := #IO;
               "VOLVO 16 09 KP8 Out" := #"KP8 Out";
           #"VOLVO 16 10":
               "VOLVO 16 10 IO" := #IO;
               "VOLVO 16 10 KP8 Out" := #"KP8 Out";
           #"VOLVO 16 11":
               "VOLVO 16 11 IO" := #IO;
               "VOLVO 16 11 KP8 Out" := #"KP8 Out";
           #"CHM 01":
               "CHM 01 IO" := #IO;
               "CHM 01 KP8 Out" := #"KP8 Out";
           #"CHM 02":
               "CHM 02 IO" := #IO;
               "CHM 02 KP8 Out" := #"KP8 Out";
           #"CHM 03":
               "CHM 03 IO" := #IO;
               "CHM 03 KP8 Out" := #"KP8 Out";
           #"CHM 04":
               "CHM 04 IO" := #IO;
               "CHM 04 KP8 Out" := #"KP8 Out";
           #"CHM 05":
               "CHM 05 IO" := #IO;
               "CHM 05 KP8 Out" := #"KP8 Out";
           #"CDO 01":
               "CDO 01 IO" := #IO;
               "CDO 01 KP8 Out" := #"KP8 Out";
           #"CDO 02":
               "CDO 02 IO" := #IO;
               "CDO 02 KP8 Out" := #"KP8 Out";
           #"CDO 03":
               "CDO 03 IO" := #IO;
               "CDO 03 KP8 Out" := #"KP8 Out";
           #"BFL 01":
               "BFL 01 IO" := #IO;
               "BFL 01 KP8 Out" := #"KP8 Out";
           #"BFL 02":
               "BFL 02 IO" := #IO;
               "BFL 02 KP8 Out" := #"KP8 Out";
           #"BFL 03":
               "BFL 03 IO" := #IO;
               "BFL 03 KP8 Out" := #"KP8 Out";
           #"LGS 01":
               "LGS 01 IO" := #IO;
               "LGS 01 KP8 Out" := #"KP8 Out";
           #"LGS 02":
               "LGS 02 IO" := #IO;
               "LGS 02 KP8 Out" := #"KP8 Out";

       END_CASE;

   END_FOR;
END_REGION
END_FUNCTION

FUNCTION "Select Stations" : Void   // FC6, SCL
{ S7_Optimized_Access := 'TRUE' }
VERSION : 0.1
   VAR_INPUT
      constants : "Constants";
      mode : Bool;   // TRUE = select; FALSE = deselect
   END_VAR
   VAR_IN_OUT
      stations : "Stations";
   END_VAR
   VAR_TEMP
      i : Int;
      stnCount : Int;
   END_VAR
   VAR CONSTANT
      stationCount : Int := 22;
   END_VAR
BEGIN
   REGION "GET STATION COUNT"
       #stnCount := #constants.stationCount - 1;
   END_REGION

   REGION "SELECT STATIONS"
       FOR #i := 0 TO #stnCount DO
           #stations.current[#i].settings.selected := #mode;
       END_FOR;
   END_REGION
END_FUNCTION

FUNCTION "Select Buttons" : Void   // FC8, SCL
{ S7_Optimized_Access := 'TRUE' }
VERSION : 0.1
   VAR_INPUT
      constants : "Constants";
      mode : Bool;   // TRUE = select; FALSE = deselect
   END_VAR
   VAR_IN_OUT
      stations : "Stations";
   END_VAR
   VAR_TEMP
      btnCount : Int;
      i : Int;
      j : Int;
      selected : Bool;
      stnCount : Int;
   END_VAR
   VAR CONSTANT
      buttonCount : Int := 5;
   END_VAR
BEGIN
   REGION "COPY TO LOCAL"
       #btnCount := #constants.buttonCount - 1;
       #stnCount := #constants.stationCount - 1;
   END_REGION

   REGION "SELECT BUTTONS"
       FOR #i := 0 TO #stnCount DO

           REGION "SELCT ALL BUTTONS ON SELECTED STATION"
               #selected := #stations.current[#i].settings.selected;
               IF #selected THEN

                   REGION "LOOP THROUGH BUTTONS"
                       FOR #j := 0 TO #btnCount DO
                           #stations.current[#i].settings.btnSelection[#j] := #mode;
                       END_FOR;
                   END_REGION

               END_IF;
           END_REGION

       END_FOR;
   END_REGION
END_FUNCTION

FUNCTION "Animate Bool" : USInt   // FC9, SCL
{ S7_Optimized_Access := 'TRUE' }
VERSION : 0.1
   VAR_INPUT
      colorTrue : USInt;
      colorFalse : USInt;
      evalSignal : Bool;
   END_VAR
   VAR_TEMP
      animate : USInt;
   END_VAR
BEGIN
   REGION "FALSE COLOR"
       IF NOT #evalSignal THEN
           #animate := #colorFalse;
       END_IF;
   END_REGION

   REGION "TRUE COLOR"
       IF #evalSignal THEN
           #animate := #colorTrue;
       END_IF;
   END_REGION

   REGION "FUNCTION RETURN"
       #"Animate Bool" := #animate;
   END_REGION
END_FUNCTION

FUNCTION "WString to Time" : Time   // FC10, SCL
{ S7_Optimized_Access := 'TRUE' }
VERSION : 0.1
   VAR_INPUT
      WString : WString;
   END_VAR
   VAR_TEMP
      Count : UInt;
      "DInt Box" : DInt;
      "String Box" : WString [5];
      "Time Box" : Time;
      "WChar Array" : Array[0..4] of WChar;
   END_VAR
   VAR CONSTANT
      "ms/(10 hr)" : DInt := 36000000;
      "ms/hr" : DInt := 3600000;
      "ms/(10 min)" : DInt := 600000;
      "ms/min" : DInt := 60000;
      "ms/(10 sec)" : DInt := 10000;
      "ms/sec" : DInt := 1000;
   END_VAR
BEGIN
   REGION EXPLODE INPUT

       #"String Box" := #WString;
       IF #"String Box" = WSTRING#'' THEN
           #"String Box" := WSTRING#'00:00';
       END_IF;

       Strg_TO_Chars(Strg := #"String Box",
                     pChars := 0,
                     Cnt => #Count,
                     Chars := #"WChar Array");

   END_REGION

   REGION CONVERT ARRAY ELEMENTS TO TIME

       // 10S OF MINUTES
       #"DInt Box" := WCHAR_TO_DINT(IN := #"WChar Array"[0]) - 16#30;
       #"Time Box" := #"Time Box" + #"DInt Box" * #"ms/(10 min)";

       // MINUTES
       #"DInt Box" := WCHAR_TO_DINT(IN := #"WChar Array"[1]) - 16#30;
       #"Time Box" := #"Time Box" + #"DInt Box" * #"ms/min";

       // 10S OF SECONDS
       #"DInt Box" := WCHAR_TO_DINT(IN := #"WChar Array"[3]) - 16#30;
       #"Time Box" := #"Time Box" + #"DInt Box" * #"ms/(10 sec)";

       // SECONDS
       #"DInt Box" := WCHAR_TO_DINT(IN := #"WChar Array"[4]) - 16#30;
       #"Time Box" := #"Time Box" + #"DInt Box" * #"ms/sec";

   END_REGION


   REGION RETURN VALUE

       #"WString to Time" := #"Time Box";

   END_REGION
END_FUNCTION

FUNCTION "Get Part Call Row Number" : Int   // FC11, SCL
{ S7_Optimized_Access := 'TRUE' }
VERSION : 0.1
   VAR_INPUT
      constants : "Constants";
   END_VAR
   VAR_IN_OUT
      partCall : "Part Call Screen";
   END_VAR
   VAR_TEMP
      hmiRows : Int;
      i : Int;
      selectedRow : Int;
   END_VAR
BEGIN
   REGION "GET NUMBER OF HMI ROWS"
       #hmiRows := #constants.hmiRowCount - 1;
   END_REGION

   REGION "LOOP THROUGH HMI ROWS
       FOR #i := 0 TO #hmiRows DO

           REGION "FIND SELECTED ROW"
               IF #partCall.current[#i].pbSelection.actuate THEN
                   // selected row as int
                   #selectedRow := #i + 1;
                   EXIT;
               END_IF;
           END_REGION

       END_FOR;
   END_REGION

   REGION "RETURN ROW NUMBER"
       #"Get Part Call Row Number" := #selectedRow;
   END_REGION
END_FUNCTION

FUNCTION "Address to Station and Button" : Void   // FC12, SCL
{ S7_Optimized_Access := 'TRUE' }
VERSION : 0.1
   VAR_INPUT
      address : UInt;
   END_VAR
   VAR_OUTPUT
      station : UInt;
      button : UInt;
   END_VAR
BEGIN
   #station := #address / 10;
   #button := #address MOD 10;
END_FUNCTION

FUNCTION "WString Timer to Real" : Real   // FC13, SCL
{ S7_Optimized_Access := 'TRUE' }
VERSION : 0.1
   VAR_INPUT
      wstring : WString;
   END_VAR
   VAR CONSTANT
      msPerSec : Real := 1000.0;
   END_VAR
BEGIN
   #"WString Timer to Real" := DINT_TO_REAL(TIME_TO_DINT("WString to Time"(#wstring))) / #msPerSec;
END_FUNCTION

FUNCTION "Real to WString Timer" : WString   // FC14, SCL
{ S7_Optimized_Access := 'TRUE' }
VERSION : 0.1
   VAR_INPUT
      realVal : Real;
   END_VAR
   VAR CONSTANT
      msPerSec : Real := 1000.0;
   END_VAR
BEGIN
   #"Real to WString Timer" := "Time to WString"(DINT_TO_TIME(REAL_TO_DINT(#realVal * #msPerSec)));
END_FUNCTION

ORGANIZATION_BLOCK "Main"   // OB1, LAD, ProgramCycle
TITLE = "Main Program Sweep (Cycle)"
{ S7_Optimized_Access := 'TRUE' }
VERSION : 0.1
   VAR_INPUT
      Initial_Call : Bool;   // Initial call of this OB
      Remanence : Bool;   // =True, if remanent data are available
   END_VAR
BEGIN

